PROGRAM MAINSafety
VAR CONSTANT
	sNetID: T_AmsNetId := '10.24.33.33.2.1'; // EtherCAT Master AMS NetID
END_VAR
VAR
	(* I/O *)
	bEnable 			AT %I*	: BOOL; (* Pozwolenie na prace z SAFETY ESTOP *)
	stSAFETYGroupIO				: ST_SAFETYGroupIO;
	fbSAFETY_AutoGroupErrACK	: FB_SAFETY_AutoGroupErrACK;
	(* HW diagnostic *)
	fbEL1904_DiagnosticData		: FB_EL1904_DiagnosticData;
	stEL1904_DiagnosticData		: ST_EL1904_DiagnosticData;
	fbEL2904_DiagnosticData		: FB_EL2904_DiagnosticData;
	stEL2904_DiagnosticData		: ST_EL2904_DiagnosticData;
	fbEL6900_DiagnosticData		: FB_EL6900_DiagnosticData;
	stEL6900_DiagnosticData		: ST_EL6900_DiagnosticData;
	(* SAFETY project diagnostic *)
	fbEL6900_StatusData			: FB_EL6900_StatusData;
	stEL6900_StatusData			: ST_EL6900_StatusData;
	(* FBs conversion *)
	stSAFETY_FBESTOP			: ST_SAFETY_FBESTOP;
	stSAFETY_FBTwoHand			: ST_SAFETY_FBTWOHAND;
	stSAFETY_FBRS				: ST_SAFETY_FBRS;
	stSAFETY_FBTOF				: ST_SAFETY_FBTOF;
	stSAFETY_FBOPMODE			: ST_SAFETY_FBOPMODE;
	stSAFETY_FBMUTING			: ST_SAFETY_FBMUTING;
	stSAFETY_FBMON				: ST_SAFETY_FBMON;
	stSAFETY_FBDECOUPLE			: ST_SAFETY_FBDECOUPLE;
	stSAFETY_FBAND				: ST_SAFETY_FBAND;
	stSAFETY_FBOR				: ST_SAFETY_FBOR;
	(* Other *)
	tonDelay					: TON;
	rtInit						: R_TRIG;
	ftEL1904DiagEnd				: F_TRIG;
	ftEL2904DiagEnd				: F_TRIG;
	ftEL6900DiagEnd				: F_TRIG;
	ftEL6900StatusEnd			: F_TRIG;
END_VAR

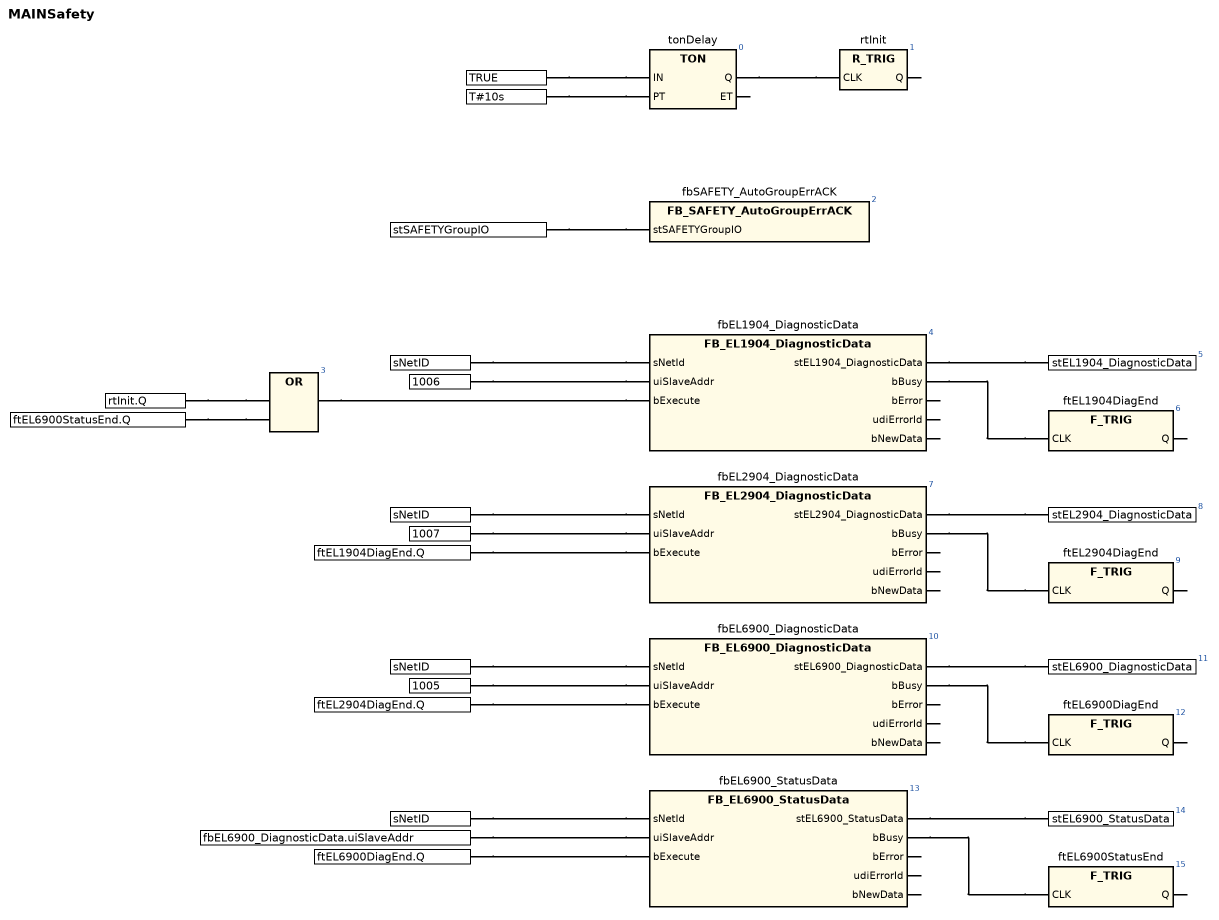
tonDelay(IN := TRUE, PT := T#10s); // TON
rtInit(CLK := tonDelay.Q); // R_TRIG
fbSAFETY_AutoGroupErrACK(stSAFETYGroupIO := stSAFETYGroupIO); // FB_SAFETY_AutoGroupErrACK
fbEL1904_DiagnosticData(sNetId := sNetID, uiSlaveAddr := 1006, bExecute := rtInit.Q OR ftEL6900StatusEnd.Q); // FB_EL1904_DiagnosticData
stEL1904_DiagnosticData := fbEL1904_DiagnosticData.stEL1904_DiagnosticData;
ftEL1904DiagEnd(CLK := fbEL1904_DiagnosticData.bBusy); // F_TRIG
fbEL2904_DiagnosticData(sNetId := sNetID, uiSlaveAddr := 1007, bExecute := ftEL1904DiagEnd.Q); // FB_EL2904_DiagnosticData
stEL2904_DiagnosticData := fbEL2904_DiagnosticData.stEL2904_DiagnosticData;
ftEL2904DiagEnd(CLK := fbEL2904_DiagnosticData.bBusy); // F_TRIG
fbEL6900_DiagnosticData(sNetId := sNetID, uiSlaveAddr := 1005, bExecute := ftEL2904DiagEnd.Q); // FB_EL6900_DiagnosticData
stEL6900_DiagnosticData := fbEL6900_DiagnosticData.stEL6900_DiagnosticData;
ftEL6900DiagEnd(CLK := fbEL6900_DiagnosticData.bBusy); // F_TRIG
fbEL6900_StatusData(
    sNetId := sNetID,
    uiSlaveAddr := fbEL6900_DiagnosticData.uiSlaveAddr,
    bExecute := ftEL6900DiagEnd.Q); // FB_EL6900_StatusData
stEL6900_StatusData := fbEL6900_StatusData.stEL6900_StatusData;
ftEL6900StatusEnd(CLK := fbEL6900_StatusData.bBusy); // F_TRIG

END_PROGRAM

(* stored: Version 1.1.0.1, ProductVersion 3.1.4022.12
   POU MAINSafety: Id {38e4432d-32aa-4423-89df-562f3e63bdd3}, SpecialFunc None *)
